TYPE state_transition_commands_t :
(
	Shutdown,
	SwitchOn,
	SwitchOnEnOP,
	DisableVolt,
	QuickStop,
	DisableOP,
	EnableOP,
	FaultReset
);
END_TYPE

(* stored: Version 1.1.0.1, ProductVersion 3.1.4024.12
   DUT state_transition_commands_t: Id {d09dfb61-40a1-4c2d-8d77-0856c1a88186} *)
